{attribute 'qualified_only'}
{attribute 'strict'}
TYPE E_Event :
(
	SwitchOn := 0,
	SwitchOff := 1,
	HeatIsRequested := 2,
	HeatTemperaturreached := 3,
	CooledDown := 4,
	Confirmed := 5
);
END_TYPE

(* stored: Version 1.1.0.1
   DUT E_Event: Id {5974e92a-1925-4467-bd7b-7d781837f1c3} *)
